FUNCTION Inc
VAR_INPUT
	In : POINTER TO DINT;
END_VAR

In^ := In^ + 1;

END_FUNCTION

(* stored: Version 1.1.0.1, ProductVersion 3.1.4024.15
   POU Inc: Id {231dae03-7c76-4d0c-af81-6666a3accebe}, SpecialFunc None *)
